{attribute 'linkalways'} 
{attribute 'no_explicit_call' := 'This FB is a CLASS and must be accessed using methods or properties'}
{attribute 'enable_dynamic_creation'}
FUNCTION_BLOCK Node_F_VN_DarkBorderObjects EXTENDS VisionNode
VAR
    ipSrcImage : _ITcVnImage;
    ipDestImage : _ITcVnImage;
    hrPrev : _HRESULT(S_OK);
	hresult : _HRESULT(S_OK);
END_VAR

METHOD PUBLIC  Clone : I_Node
VAR
	pNode : POINTER TO Node_F_VN_DarkBorderObjects;
END_VAR
pNode := __NEW(Node_F_VN_DarkBorderObjects);
Clone := pNode^;
END_METHOD

METHOD FB_init : BOOL
VAR_INPUT
	bInitRetains : BOOL; // if TRUE, the retain variables are initialized (warm start / cold start)
	bInCopyCode : BOOL;  // if TRUE, the instance afterwards gets moved into the copy code (online change)
END_VAR
AddInput('ipSrcImage', ipSrcImage);
AddInput('hrPrev', hrPrev);
AddOutput('ipDestImage', ipDestImage);
AddOutput('hresult',hresult);
END_METHOD

METHOD PROTECTED OnExecute : HRESULT
hresult.Value := F_VN_DarkBorderObjects(
    ipSrcImage := ipSrcImage.Value,
	ipDestImage := ipDestImage.Value,
	hrPrev:= hrPrev.Value);
END_METHOD

METHOD PUBLIC PreExecutionCheck
VAR_INPUT
	Check : I_PreExecutionChecks;
END_VAR
IF FAILED(hrPrev.Value) THEN
    RETURN;
END_IF

Check.IsTrue(ipSrcImage.IsValid, 'ipSrcImage must contain an image');
Check.IsTrue(ipSrcImage.HasChannelCount(1), 'ipSrcImage must have 1 channel');

Check.IsTrue((ipSrcImage.IsPixelDepth(8)  OR
              ipSrcImage.IsPixelDepth(16) OR
              ipSrcImage.IsPixelDepth(32) OR
              ipSrcImage.IsPixelDepth(64)), 'ipSrcImage must have 8, 16, 32 or 64 bit pixel depth');
END_METHOD

END_FUNCTION_BLOCK

(* stored: Version 1.1.0.1, ProductVersion 3.1.4024.13
   POU Node_F_VN_DarkBorderObjects: Id {d7e4e079-d160-05a7-2f0d-1afa04d7b1e6}, SpecialFunc None
   Folder Constructor: Id {530464f7-e893-0289-389b-a9274cfbf53f}
   Method Clone: Id {116eee86-de42-0feb-1260-33b1d66cde3a}
   Method FB_init: Id {4b04317a-55e0-0989-3970-4d6bc81aca77}
   Method OnExecute: Id {76acbb58-1a21-0a65-273a-28f8af712319}
   Method PreExecutionCheck: Id {a0fdcff5-8e13-01c6-3302-088fd68bf49f} *)
